(* Logix 5000 project; controller CompactLogix Emulate 5570 rev 16.42; software revision 16.03 *)

TASK MainTask (periodic, rate 50 ms, priority 10, watchdog 500 ms) : MainProgram

MODULES
   Local : Emulate 5570 (ICP 1, rev 16.42)
       : 1756-IA16 (ICP 2, rev 2.1, Input RPI 20 ms)
       : vendor 1 type 7 code 13 (ICP 3, rev 2.1, Output RPI 20 ms)
END_MODULES

PROGRAM MainProgram   (* main routine MainRoutine *)
VAR
   Area : REAL;   // cumulative area calculation
   deltaA : REAL;   // per-scan area added
   iscan : REAL;   // [0:64]
   L : REAL;   // Level parameter in loop
   L0 : REAL;   // Actual level, [-32.0:+32.0]
   R : REAL;   // Tank radius
   tttN : REAL;   // Scaling factor in loop, 2**N
END_VAR

ROUTINE MainRoutine   (* ladder *)
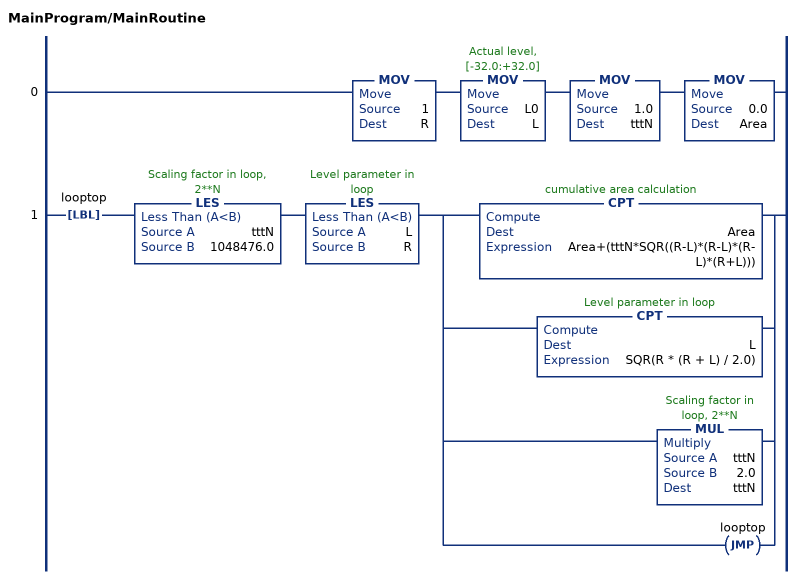
   0: MOV(1,R)MOV(L0,L)MOV(1.0,tttN)MOV(0.0,Area);
   1: LBL(looptop)LES(tttN,1048476.0)LES(L,R)[CPT(Area,Area+(tttN*SQR((R-L)*(R-L)*(R-L)*(R+L)))) ,CPT(L,SQR(R * (R + L) / 2.0)) ,MUL(tttN,2.0,tttN) ,JMP(looptop) ];
END_ROUTINE
END_PROGRAM
